(* Logix 5000 project; controller DispersionPlc vendor 1 type 14 code 108 rev 34.11; software revision 34.01; part 18 of 22 *)
(* tags used below, declared in another part *)
   _JISdebug : DINT;
   constant : REAL;
   Estop_Disp : ALIAS FOR Local:3:I.Data.1;
   FilterChangePB : BOOL;
   FIT_4302_1 : AStd_AnalogInput;
   FQIC_4302_11_CurrentTrasferredLb : DINT;
   FQIC_4302_11_Reset : BOOL;
   FQIC_4302_11_TransferSetpoint : DINT;
   FQIC_4302_11_TransferStopValueLb : DINT;
   GenPurp : AStd_GeneralPurp;
   LAH_4302_11 : BOOL;   // Truck Loading Level Alarm High Probe
   LAH_S4352_1 : ALIAS FOR Local:1:I.Data[27].13;
   resetTimer : BOOL;
   ROC_SP : REAL;
   ROC_SP_10min : REAL;
   S4352_Phase_Circulation : AStd_PLI;
   S4352_Phase_Packaging_Transfer : AStd_PLI;
   S4352_Phase_TT_Transfer : AStd_PLI;
   S52TransferCompletePB : BOOL;
   SP : REAL;
   SV_4302_1 : AStd_VlvOC;
   SV_S52_2 : AStd_VlvOC;
   T4302_Phase_S52_Transfer : AStd_PLI;
   T4302_Phase_S52_Transfer_AOI : AStd_PLI_AOI;
   T4302_Phase_TT_Transfer : AStd_PLI;
   T4302_Phase_TT_Transfer_AOI : AStd_PLI_AOI;
   T4302_PhaseAgitation : AStd_PLI;
   T4302_PhaseAgitation_AOI : AStd_PLI_AOI;
   T4302_PhaseTempControl : AStd_PLI;
   T4302_PhaseTempControl_AOI : AStd_PLI_AOI;
   T4302_RampControl : BOOL;
   T4302_RampControl_ONS : BOOL;
   T4302_RampControl_ONS_2 : BOOL;
   T4302_RampControlTOn : TIMER;
   T4302TruckTransferCompletePB : BOOL;
   TCV_4302_1 : AStd_VlvModulating;
   TCV_4302_2 : AStd_VlvModulating;
   TCV_4302_2_Mode : SINT;
   TE_4302A : ALIAS FOR Local:8:I.Ch5Data;
   TempChange : REAL;
   TIC_4302_1 : AStd_PIDInterface;
   TIC_4302_1_AOI : AStd_PIDInterface_AOI;
   TIC_4302_1_PID : PID_ENHANCED;
   TIC_4302_4C : AStd_PIDInterface;
   TIC_4302_4C_AOI : AStd_PIDInterface_AOI;
   TIC_4302_4C_PID : PID_ENHANCED;
   TIC_4302_4H : AStd_PIDInterface;
   TIC_4302_4H_AOI : AStd_PIDInterface_AOI;
   TIC_4302_4H_PID : PID_ENHANCED;
   TIT_4302_1 : AStd_AnalogInput;
   TIT_4302_4 : AStd_AnalogInput;
   VFD_4302_1 : AStd_VFD;
   VFD_P_4302_2 : AStd_VFD;
   WIT_4302_1 : AStd_AnalogInput;
   XV_4302_12 : AStd_VlvOC;
   XV_4302_13 : AStd_VlvOC;
   XV_4302_5 : AStd_VlvOC;
   XV_4302_6 : AStd_VlvOC;
   XV_S52_1 : AStd_VlvOC;
   XV_S52_2 : AStd_VlvOC;
(* Unit_T4302, continued *)

ROUTINE Phase_Agitation   (* ladder *)
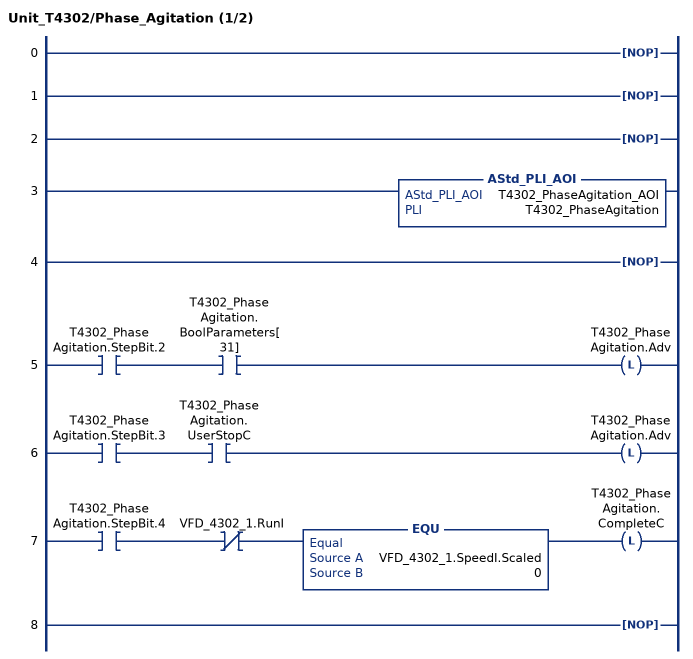
   0: NOP();
   1: NOP();
   2: NOP();
   3: AStd_PLI_AOI(T4302_PhaseAgitation_AOI,T4302_PhaseAgitation);
   4: NOP();
   5: XIC(T4302_PhaseAgitation.StepBit.2)XIC(T4302_PhaseAgitation.BoolParameters[31])OTL(T4302_PhaseAgitation.Adv);
   6: XIC(T4302_PhaseAgitation.StepBit.3)XIC(T4302_PhaseAgitation.UserStopC)OTL(T4302_PhaseAgitation.Adv);
   7: XIC(T4302_PhaseAgitation.StepBit.4)XIO(VFD_4302_1.RunI)EQU(VFD_4302_1.SpeedI.Scaled,0)OTL(T4302_PhaseAgitation.CompleteC);
   8: NOP();
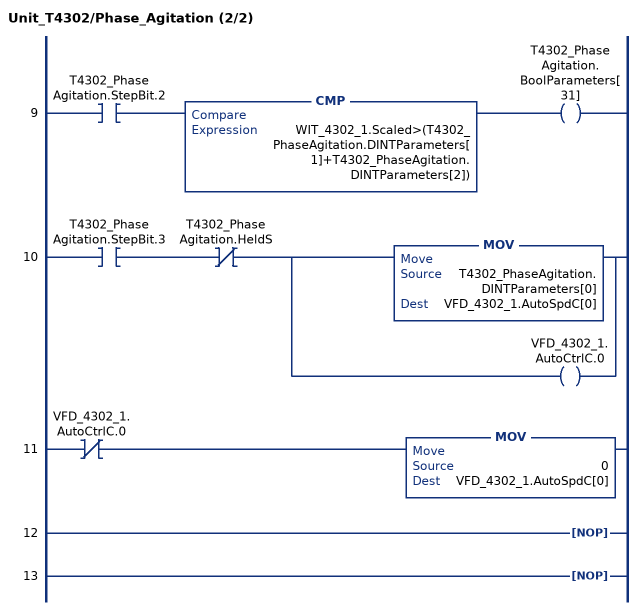
   9: XIC(T4302_PhaseAgitation.StepBit.2)CMP(WIT_4302_1.Scaled>(T4302_PhaseAgitation.DINTParameters[1]+T4302_PhaseAgitation.DINTParameters[2]))OTE(T4302_PhaseAgitation.BoolParameters[31]);
   10: XIC(T4302_PhaseAgitation.StepBit.3)XIO(T4302_PhaseAgitation.HeldS)[MOV(T4302_PhaseAgitation.DINTParameters[0],VFD_4302_1.AutoSpdC[0]) ,OTE(VFD_4302_1.AutoCtrlC.0) ];
   11: XIO(VFD_4302_1.AutoCtrlC.0)MOV(0,VFD_4302_1.AutoSpdC[0]);
   12: NOP();
   13: NOP();
END_ROUTINE

ROUTINE Phase_S52_Transfer   (* ladder *)
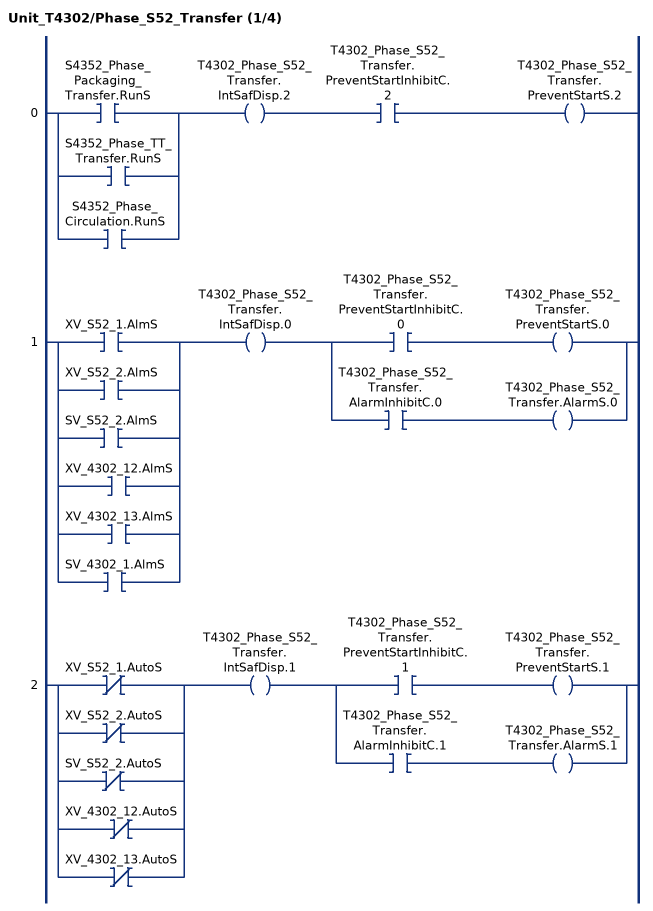
   0: [XIC(S4352_Phase_Packaging_Transfer.RunS) ,XIC(S4352_Phase_TT_Transfer.RunS) ,XIC(S4352_Phase_Circulation.RunS) ]OTE(T4302_Phase_S52_Transfer.IntSafDisp.2)XIC(T4302_Phase_S52_Transfer.PreventStartInhibitC.2)OTE(T4302_Phase_S52_Transfer.PreventStartS.2);
   1: [XIC(XV_S52_1.AlmS) ,XIC(XV_S52_2.AlmS) ,XIC(SV_S52_2.AlmS) ,XIC(XV_4302_12.AlmS) ,XIC(XV_4302_13.AlmS) ,XIC(SV_4302_1.AlmS) ]OTE(T4302_Phase_S52_Transfer.IntSafDisp.0)[XIC(T4302_Phase_S52_Transfer.PreventStartInhibitC.0) OTE(T4302_Phase_S52_Transfer.PreventStartS.0) ,XIC(T4302_Phase_S52_Transfer.AlarmInhibitC.0) OTE(T4302_Phase_S52_Transfer.AlarmS.0) ];
   2: [XIO(XV_S52_1.AutoS) ,XIO(XV_S52_2.AutoS) ,XIO(SV_S52_2.AutoS) ,XIO(XV_4302_12.AutoS) ,XIO(XV_4302_13.AutoS) ]OTE(T4302_Phase_S52_Transfer.IntSafDisp.1)[XIC(T4302_Phase_S52_Transfer.PreventStartInhibitC.1) OTE(T4302_Phase_S52_Transfer.PreventStartS.1) ,XIC(T4302_Phase_S52_Transfer.AlarmInhibitC.1) OTE(T4302_Phase_S52_Transfer.AlarmS.1) ];
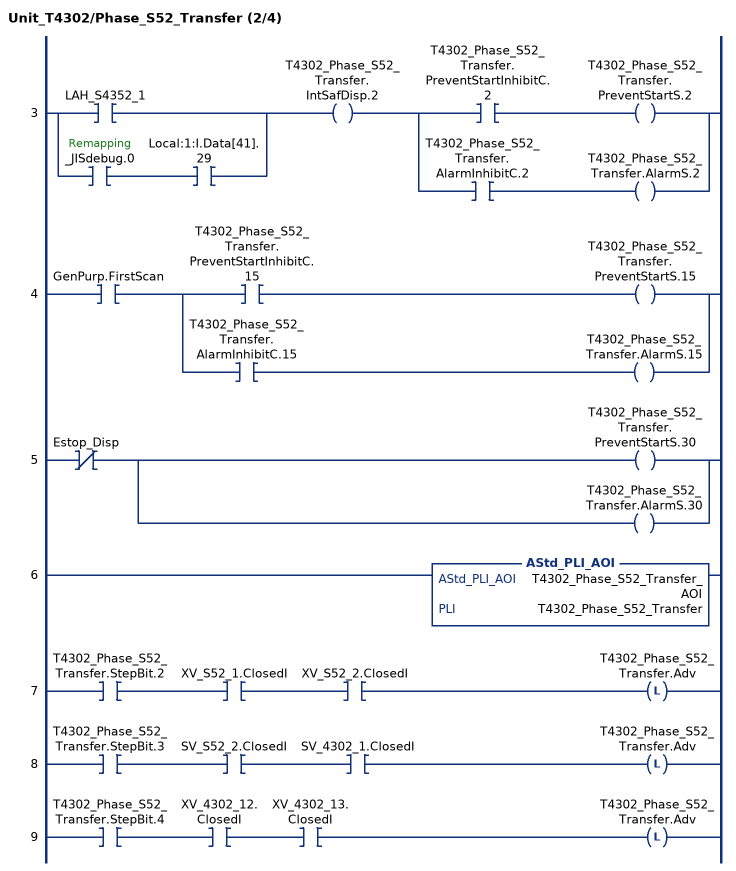
   3: [XIC(LAH_S4352_1) ,XIC(_JISdebug.0) XIC(Local:1:I.Data[41].29) ]OTE(T4302_Phase_S52_Transfer.IntSafDisp.2)[XIC(T4302_Phase_S52_Transfer.PreventStartInhibitC.2) OTE(T4302_Phase_S52_Transfer.PreventStartS.2) ,XIC(T4302_Phase_S52_Transfer.AlarmInhibitC.2) OTE(T4302_Phase_S52_Transfer.AlarmS.2) ];
   4: XIC(GenPurp.FirstScan)[XIC(T4302_Phase_S52_Transfer.PreventStartInhibitC.15) OTE(T4302_Phase_S52_Transfer.PreventStartS.15) ,XIC(T4302_Phase_S52_Transfer.AlarmInhibitC.15) OTE(T4302_Phase_S52_Transfer.AlarmS.15) ];
   5: XIO(Estop_Disp)[OTE(T4302_Phase_S52_Transfer.PreventStartS.30) ,OTE(T4302_Phase_S52_Transfer.AlarmS.30) ];
   6: AStd_PLI_AOI(T4302_Phase_S52_Transfer_AOI,T4302_Phase_S52_Transfer);
   7: XIC(T4302_Phase_S52_Transfer.StepBit.2)XIC(XV_S52_1.ClosedI)XIC(XV_S52_2.ClosedI)OTL(T4302_Phase_S52_Transfer.Adv);
   8: XIC(T4302_Phase_S52_Transfer.StepBit.3)XIC(SV_S52_2.ClosedI)XIC(SV_4302_1.ClosedI)OTL(T4302_Phase_S52_Transfer.Adv);
   9: XIC(T4302_Phase_S52_Transfer.StepBit.4)XIC(XV_4302_12.ClosedI)XIC(XV_4302_13.ClosedI)OTL(T4302_Phase_S52_Transfer.Adv);
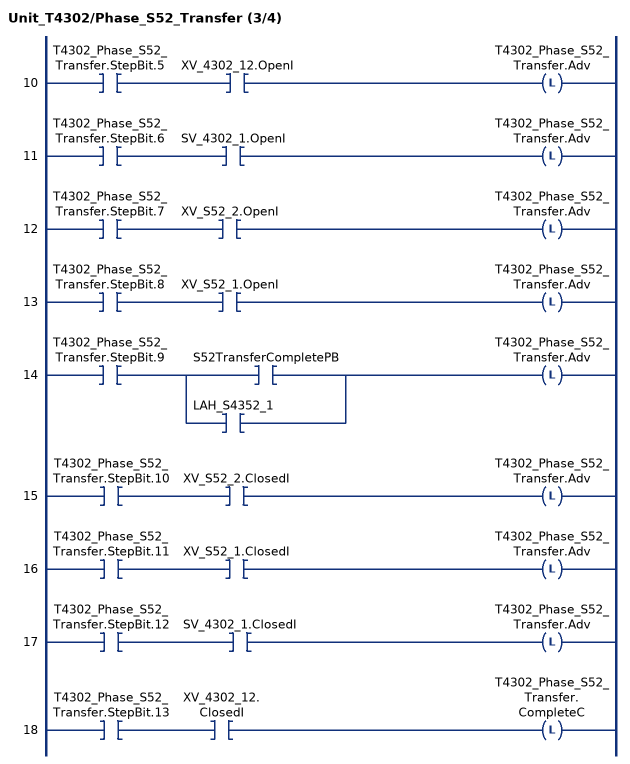
   10: XIC(T4302_Phase_S52_Transfer.StepBit.5)XIC(XV_4302_12.OpenI)OTL(T4302_Phase_S52_Transfer.Adv);
   11: XIC(T4302_Phase_S52_Transfer.StepBit.6)XIC(SV_4302_1.OpenI)OTL(T4302_Phase_S52_Transfer.Adv);
   12: XIC(T4302_Phase_S52_Transfer.StepBit.7)XIC(XV_S52_2.OpenI)OTL(T4302_Phase_S52_Transfer.Adv);
   13: XIC(T4302_Phase_S52_Transfer.StepBit.8)XIC(XV_S52_1.OpenI)OTL(T4302_Phase_S52_Transfer.Adv);
   14: XIC(T4302_Phase_S52_Transfer.StepBit.9)[XIC(S52TransferCompletePB) ,XIC(LAH_S4352_1) ]OTL(T4302_Phase_S52_Transfer.Adv);
   15: XIC(T4302_Phase_S52_Transfer.StepBit.10)XIC(XV_S52_2.ClosedI)OTL(T4302_Phase_S52_Transfer.Adv);
   16: XIC(T4302_Phase_S52_Transfer.StepBit.11)XIC(XV_S52_1.ClosedI)OTL(T4302_Phase_S52_Transfer.Adv);
   17: XIC(T4302_Phase_S52_Transfer.StepBit.12)XIC(SV_4302_1.ClosedI)OTL(T4302_Phase_S52_Transfer.Adv);
   18: XIC(T4302_Phase_S52_Transfer.StepBit.13)XIC(XV_4302_12.ClosedI)OTL(T4302_Phase_S52_Transfer.CompleteC);
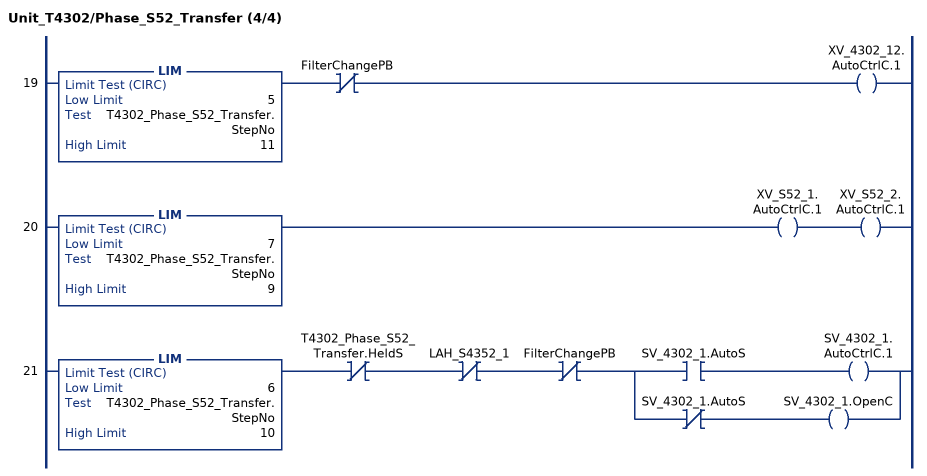
   19: LIM(5,T4302_Phase_S52_Transfer.StepNo,11)XIO(FilterChangePB)OTE(XV_4302_12.AutoCtrlC.1);
   20: LIM(7,T4302_Phase_S52_Transfer.StepNo,9)OTE(XV_S52_1.AutoCtrlC.1)OTE(XV_S52_2.AutoCtrlC.1);
   21: LIM(6,T4302_Phase_S52_Transfer.StepNo,10)XIO(T4302_Phase_S52_Transfer.HeldS)XIO(LAH_S4352_1)XIO(FilterChangePB)[XIC(SV_4302_1.AutoS) OTE(SV_4302_1.AutoCtrlC.1) ,XIO(SV_4302_1.AutoS) OTE(SV_4302_1.OpenC) ];
END_ROUTINE

ROUTINE Phase_TempControl   (* ladder *)
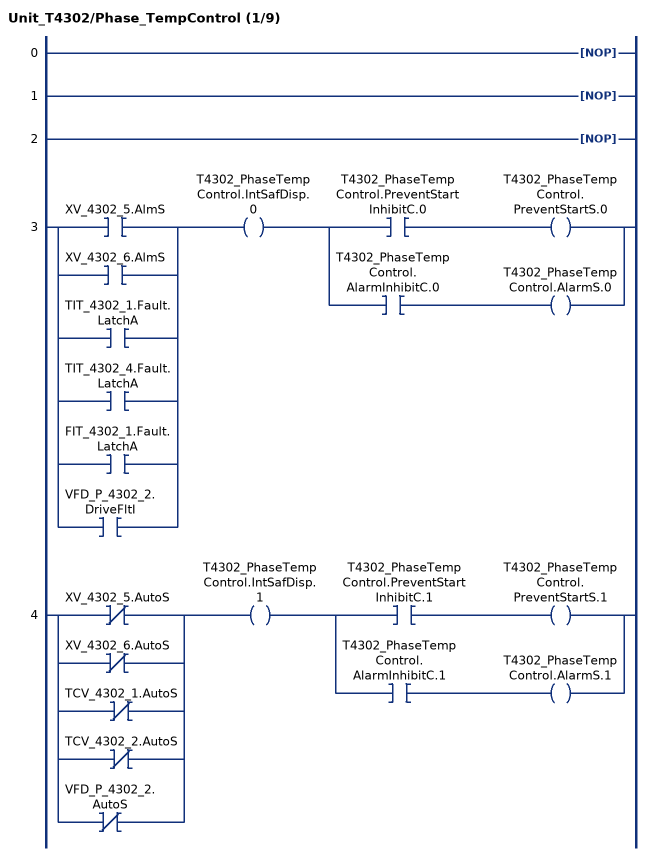
   0: NOP();
   1: NOP();
   2: NOP();
   3: [XIC(XV_4302_5.AlmS) ,XIC(XV_4302_6.AlmS) ,XIC(TIT_4302_1.Fault.LatchA) ,XIC(TIT_4302_4.Fault.LatchA) ,XIC(FIT_4302_1.Fault.LatchA) ,XIC(VFD_P_4302_2.DriveFltI) ]OTE(T4302_PhaseTempControl.IntSafDisp.0)[XIC(T4302_PhaseTempControl.PreventStartInhibitC.0) OTE(T4302_PhaseTempControl.PreventStartS.0) ,XIC(T4302_PhaseTempControl.AlarmInhibitC.0) OTE(T4302_PhaseTempControl.AlarmS.0) ];
   4: [XIO(XV_4302_5.AutoS) ,XIO(XV_4302_6.AutoS) ,XIO(TCV_4302_1.AutoS) ,XIO(TCV_4302_2.AutoS) ,XIO(VFD_P_4302_2.AutoS) ]OTE(T4302_PhaseTempControl.IntSafDisp.1)[XIC(T4302_PhaseTempControl.PreventStartInhibitC.1) OTE(T4302_PhaseTempControl.PreventStartS.1) ,XIC(T4302_PhaseTempControl.AlarmInhibitC.1) OTE(T4302_PhaseTempControl.AlarmS.1) ];
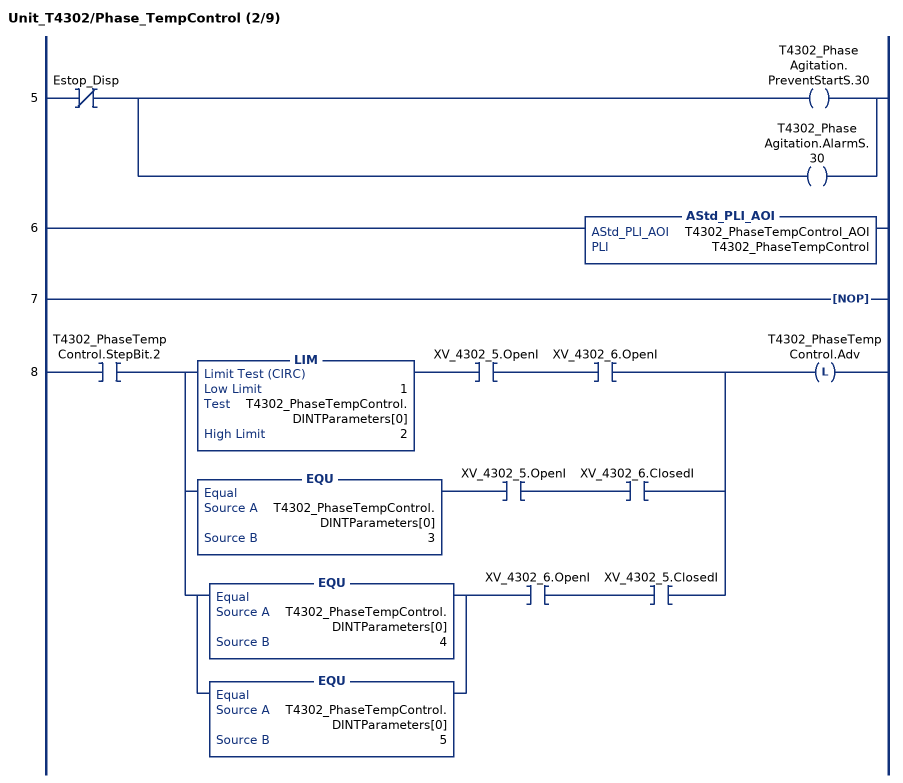
   5: XIO(Estop_Disp)[OTE(T4302_PhaseAgitation.PreventStartS.30) ,OTE(T4302_PhaseAgitation.AlarmS.30) ];
   6: AStd_PLI_AOI(T4302_PhaseTempControl_AOI,T4302_PhaseTempControl);
   7: NOP();
   8: XIC(T4302_PhaseTempControl.StepBit.2)[LIM(1,T4302_PhaseTempControl.DINTParameters[0],2) XIC(XV_4302_5.OpenI) XIC(XV_4302_6.OpenI) ,EQU(T4302_PhaseTempControl.DINTParameters[0],3) XIC(XV_4302_5.OpenI) XIC(XV_4302_6.ClosedI) ,[EQU(T4302_PhaseTempControl.DINTParameters[0],4) ,EQU(T4302_PhaseTempControl.DINTParameters[0],5) ] XIC(XV_4302_6.OpenI) XIC(XV_4302_5.ClosedI) ]OTL(T4302_PhaseTempControl.Adv);
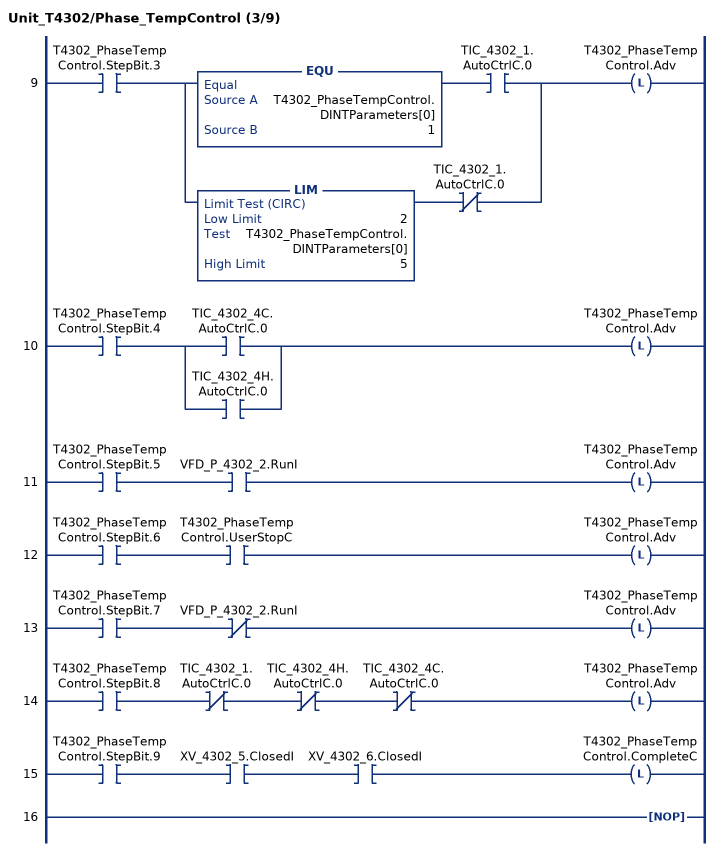
   9: XIC(T4302_PhaseTempControl.StepBit.3)[EQU(T4302_PhaseTempControl.DINTParameters[0],1) XIC(TIC_4302_1.AutoCtrlC.0) ,LIM(2,T4302_PhaseTempControl.DINTParameters[0],5) XIO(TIC_4302_1.AutoCtrlC.0) ]OTL(T4302_PhaseTempControl.Adv);
   10: XIC(T4302_PhaseTempControl.StepBit.4)[XIC(TIC_4302_4C.AutoCtrlC.0) ,XIC(TIC_4302_4H.AutoCtrlC.0) ]OTL(T4302_PhaseTempControl.Adv);
   11: XIC(T4302_PhaseTempControl.StepBit.5)XIC(VFD_P_4302_2.RunI)OTL(T4302_PhaseTempControl.Adv);
   12: XIC(T4302_PhaseTempControl.StepBit.6)XIC(T4302_PhaseTempControl.UserStopC)OTL(T4302_PhaseTempControl.Adv);
   13: XIC(T4302_PhaseTempControl.StepBit.7)XIO(VFD_P_4302_2.RunI)OTL(T4302_PhaseTempControl.Adv);
   14: XIC(T4302_PhaseTempControl.StepBit.8)XIO(TIC_4302_1.AutoCtrlC.0)XIO(TIC_4302_4H.AutoCtrlC.0)XIO(TIC_4302_4C.AutoCtrlC.0)OTL(T4302_PhaseTempControl.Adv);
   15: XIC(T4302_PhaseTempControl.StepBit.9)XIC(XV_4302_5.ClosedI)XIC(XV_4302_6.ClosedI)OTL(T4302_PhaseTempControl.CompleteC);
   16: NOP();
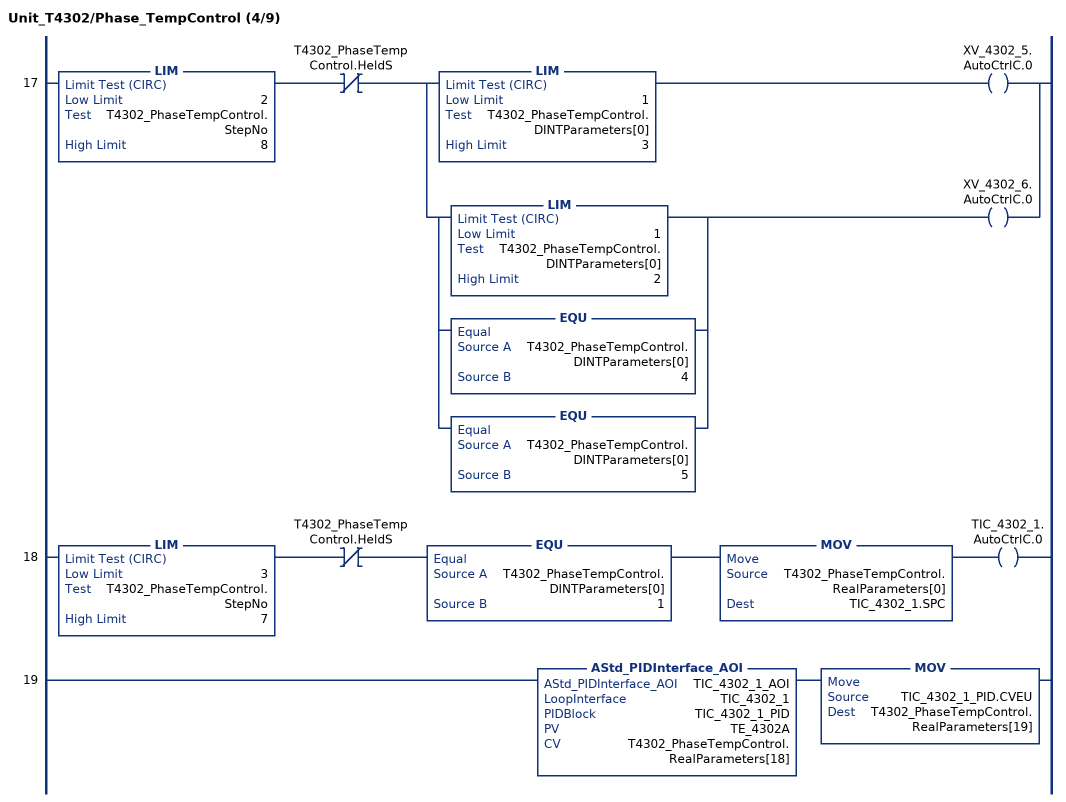
   17: LIM(2,T4302_PhaseTempControl.StepNo,8)XIO(T4302_PhaseTempControl.HeldS)[LIM(1,T4302_PhaseTempControl.DINTParameters[0],3) OTE(XV_4302_5.AutoCtrlC.0) ,[LIM(1,T4302_PhaseTempControl.DINTParameters[0],2) ,[EQU(T4302_PhaseTempControl.DINTParameters[0],4) ,EQU(T4302_PhaseTempControl.DINTParameters[0],5) ] ] OTE(XV_4302_6.AutoCtrlC.0) ];
   18: LIM(3,T4302_PhaseTempControl.StepNo,7)XIO(T4302_PhaseTempControl.HeldS)EQU(T4302_PhaseTempControl.DINTParameters[0],1)MOV(T4302_PhaseTempControl.RealParameters[0],TIC_4302_1.SPC)OTE(TIC_4302_1.AutoCtrlC.0);
   19: AStd_PIDInterface_AOI(TIC_4302_1_AOI,TIC_4302_1,TIC_4302_1_PID,TE_4302A,T4302_PhaseTempControl.RealParameters[18])MOV(TIC_4302_1_PID.CVEU,T4302_PhaseTempControl.RealParameters[19]);
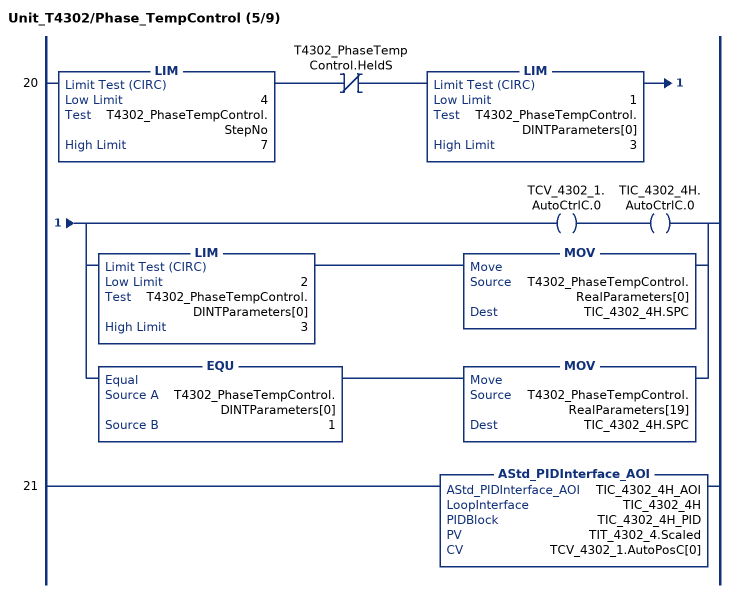
   20: LIM(4,T4302_PhaseTempControl.StepNo,7)XIO(T4302_PhaseTempControl.HeldS)LIM(1,T4302_PhaseTempControl.DINTParameters[0],3)[OTE(TCV_4302_1.AutoCtrlC.0) OTE(TIC_4302_4H.AutoCtrlC.0) ,LIM(2,T4302_PhaseTempControl.DINTParameters[0],3) MOV(T4302_PhaseTempControl.RealParameters[0],TIC_4302_4H.SPC) ,EQU(T4302_PhaseTempControl.DINTParameters[0],1) MOV(T4302_PhaseTempControl.RealParameters[19],TIC_4302_4H.SPC) ];
   21: AStd_PIDInterface_AOI(TIC_4302_4H_AOI,TIC_4302_4H,TIC_4302_4H_PID,TIT_4302_4.Scaled,TCV_4302_1.AutoPosC[0]);
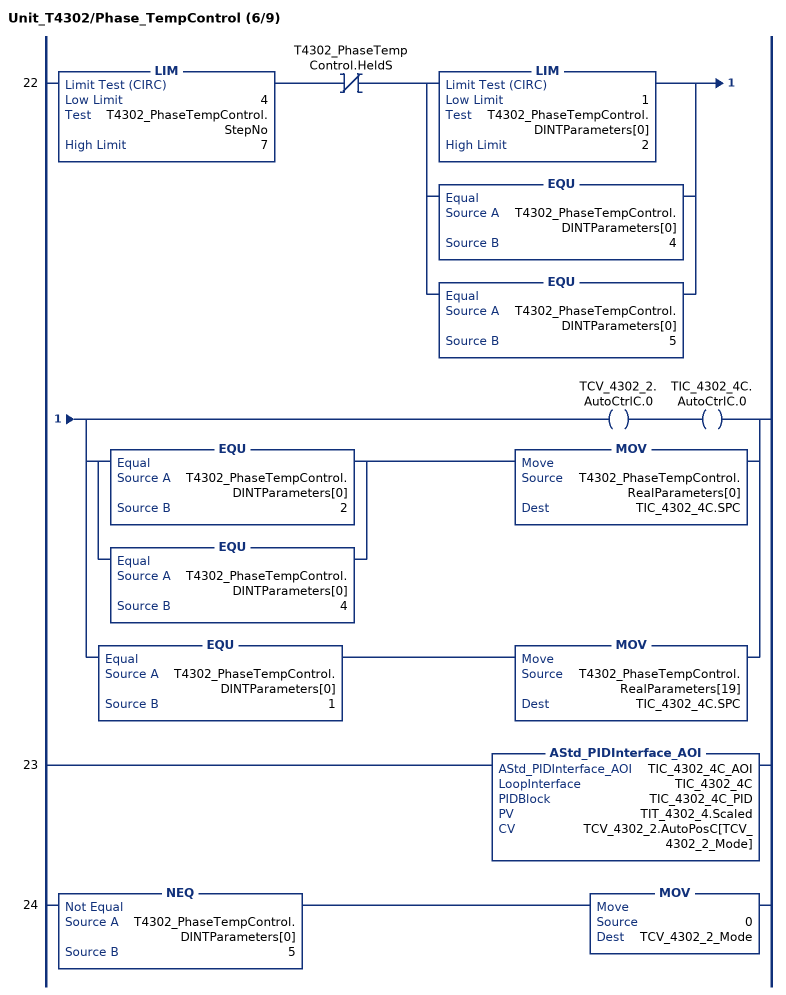
   22: LIM(4,T4302_PhaseTempControl.StepNo,7)XIO(T4302_PhaseTempControl.HeldS)[LIM(1,T4302_PhaseTempControl.DINTParameters[0],2) ,[EQU(T4302_PhaseTempControl.DINTParameters[0],4) ,EQU(T4302_PhaseTempControl.DINTParameters[0],5) ] ][OTE(TCV_4302_2.AutoCtrlC.0) OTE(TIC_4302_4C.AutoCtrlC.0) ,[EQU(T4302_PhaseTempControl.DINTParameters[0],2) ,EQU(T4302_PhaseTempControl.DINTParameters[0],4) ] MOV(T4302_PhaseTempControl.RealParameters[0],TIC_4302_4C.SPC) ,EQU(T4302_PhaseTempControl.DINTParameters[0],1) MOV(T4302_PhaseTempControl.RealParameters[19],TIC_4302_4C.SPC) ];
   23: AStd_PIDInterface_AOI(TIC_4302_4C_AOI,TIC_4302_4C,TIC_4302_4C_PID,TIT_4302_4.Scaled,TCV_4302_2.AutoPosC[TCV_4302_2_Mode]);
   24: NEQ(T4302_PhaseTempControl.DINTParameters[0],5)MOV(0,TCV_4302_2_Mode);
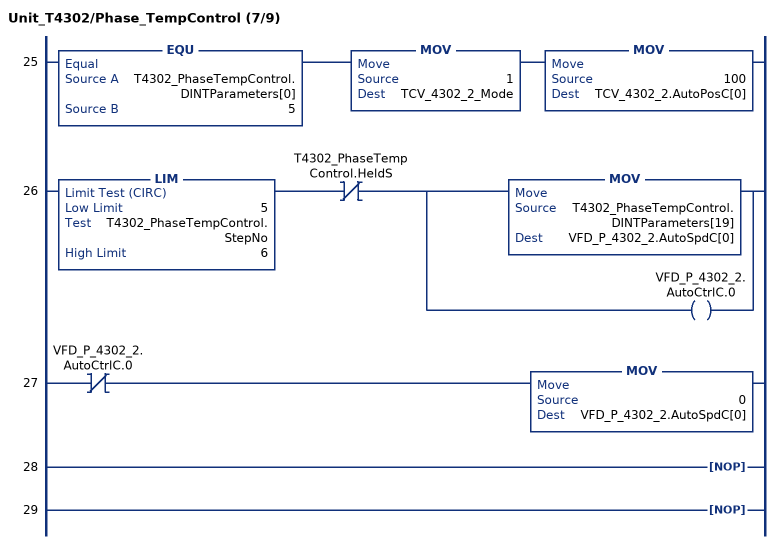
   25: EQU(T4302_PhaseTempControl.DINTParameters[0],5)MOV(1,TCV_4302_2_Mode)MOV(100,TCV_4302_2.AutoPosC[0]);
   26: LIM(5,T4302_PhaseTempControl.StepNo,6)XIO(T4302_PhaseTempControl.HeldS)[MOV(T4302_PhaseTempControl.DINTParameters[19],VFD_P_4302_2.AutoSpdC[0]) ,OTE(VFD_P_4302_2.AutoCtrlC.0) ];
   27: XIO(VFD_P_4302_2.AutoCtrlC.0)MOV(0,VFD_P_4302_2.AutoSpdC[0]);
   28: NOP();
   29: NOP();
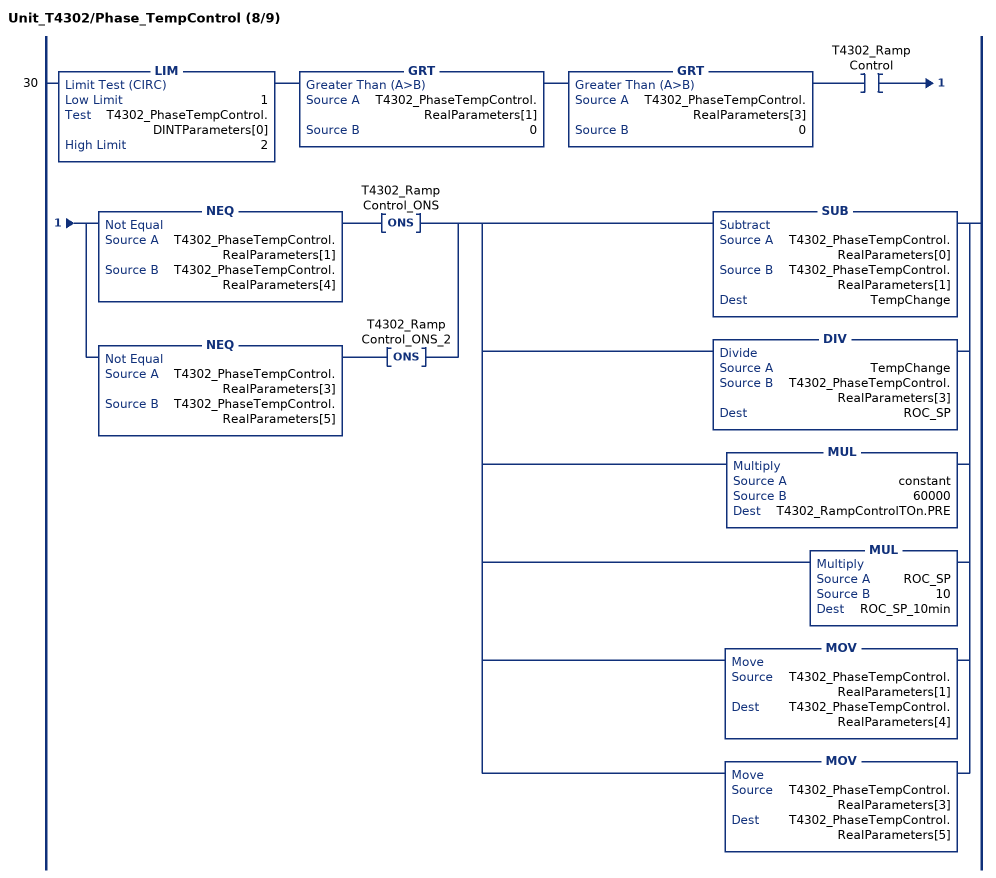
   30: LIM(1,T4302_PhaseTempControl.DINTParameters[0],2)GRT(T4302_PhaseTempControl.RealParameters[1],0)GRT(T4302_PhaseTempControl.RealParameters[3],0)XIC(T4302_RampControl)[NEQ(T4302_PhaseTempControl.RealParameters[1],T4302_PhaseTempControl.RealParameters[4]) ONS(T4302_RampControl_ONS) ,NEQ(T4302_PhaseTempControl.RealParameters[3],T4302_PhaseTempControl.RealParameters[5]) ONS(T4302_RampControl_ONS_2) ][SUB(T4302_PhaseTempControl.RealParameters[0],T4302_PhaseTempControl.RealParameters[1],TempChange) ,DIV(TempChange,T4302_PhaseTempControl.RealParameters[3],ROC_SP) ,MUL(constant,60000,T4302_RampControlTOn.PRE) ,MUL(ROC_SP,10,ROC_SP_10min) ,MOV(T4302_PhaseTempControl.RealParameters[1],T4302_PhaseTempControl.RealParameters[4]) ,MOV(T4302_PhaseTempControl.RealParameters[3],T4302_PhaseTempControl.RealParameters[5]) ];
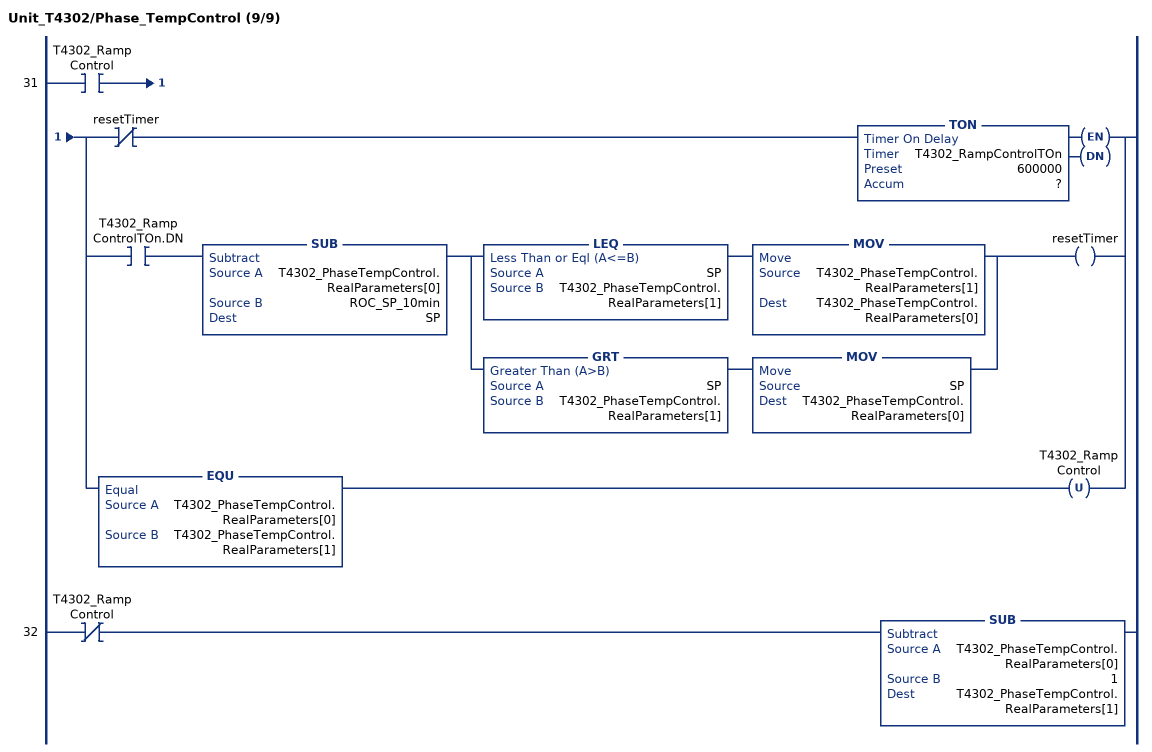
   31: XIC(T4302_RampControl)[XIO(resetTimer) TON(T4302_RampControlTOn,?,?) ,[XIC(T4302_RampControlTOn.DN) SUB(T4302_PhaseTempControl.RealParameters[0],ROC_SP_10min,SP) [LEQ(SP,T4302_PhaseTempControl.RealParameters[1]) MOV(T4302_PhaseTempControl.RealParameters[1],T4302_PhaseTempControl.RealParameters[0]) ,GRT(SP,T4302_PhaseTempControl.RealParameters[1]) MOV(SP,T4302_PhaseTempControl.RealParameters[0]) ] OTE(resetTimer) ,EQU(T4302_PhaseTempControl.RealParameters[0],T4302_PhaseTempControl.RealParameters[1]) OTU(T4302_RampControl) ] ];
   32: XIO(T4302_RampControl)SUB(T4302_PhaseTempControl.RealParameters[0],1,T4302_PhaseTempControl.RealParameters[1]);
END_ROUTINE

ROUTINE Phase_TT_Transfer   (* ladder *)
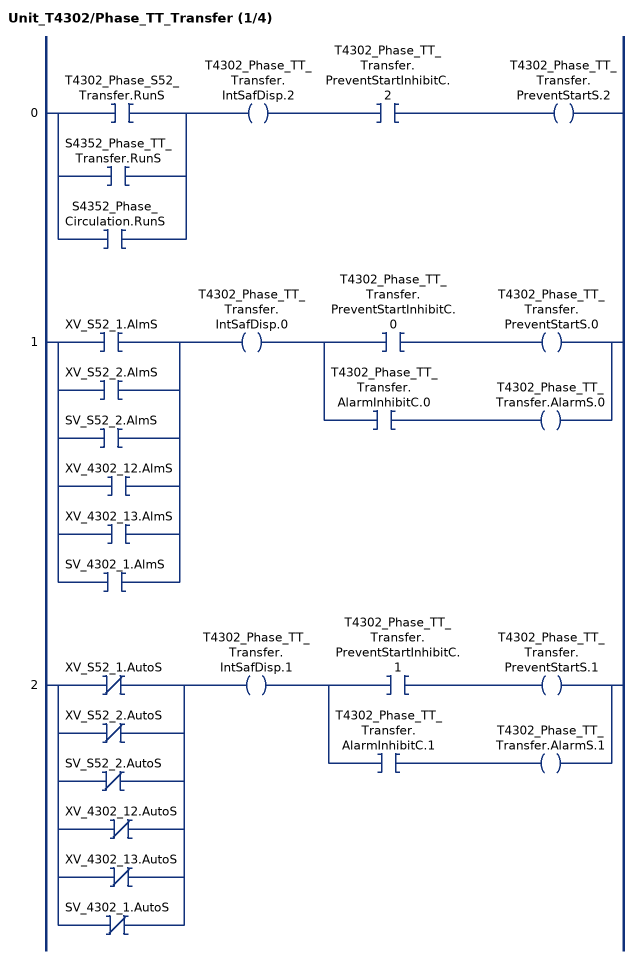
   0: [XIC(T4302_Phase_S52_Transfer.RunS) ,XIC(S4352_Phase_TT_Transfer.RunS) ,XIC(S4352_Phase_Circulation.RunS) ]OTE(T4302_Phase_TT_Transfer.IntSafDisp.2)XIC(T4302_Phase_TT_Transfer.PreventStartInhibitC.2)OTE(T4302_Phase_TT_Transfer.PreventStartS.2);
   1: [XIC(XV_S52_1.AlmS) ,XIC(XV_S52_2.AlmS) ,XIC(SV_S52_2.AlmS) ,XIC(XV_4302_12.AlmS) ,XIC(XV_4302_13.AlmS) ,XIC(SV_4302_1.AlmS) ]OTE(T4302_Phase_TT_Transfer.IntSafDisp.0)[XIC(T4302_Phase_TT_Transfer.PreventStartInhibitC.0) OTE(T4302_Phase_TT_Transfer.PreventStartS.0) ,XIC(T4302_Phase_TT_Transfer.AlarmInhibitC.0) OTE(T4302_Phase_TT_Transfer.AlarmS.0) ];
   2: [XIO(XV_S52_1.AutoS) ,XIO(XV_S52_2.AutoS) ,XIO(SV_S52_2.AutoS) ,XIO(XV_4302_12.AutoS) ,XIO(XV_4302_13.AutoS) ,XIO(SV_4302_1.AutoS) ]OTE(T4302_Phase_TT_Transfer.IntSafDisp.1)[XIC(T4302_Phase_TT_Transfer.PreventStartInhibitC.1) OTE(T4302_Phase_TT_Transfer.PreventStartS.1) ,XIC(T4302_Phase_TT_Transfer.AlarmInhibitC.1) OTE(T4302_Phase_TT_Transfer.AlarmS.1) ];
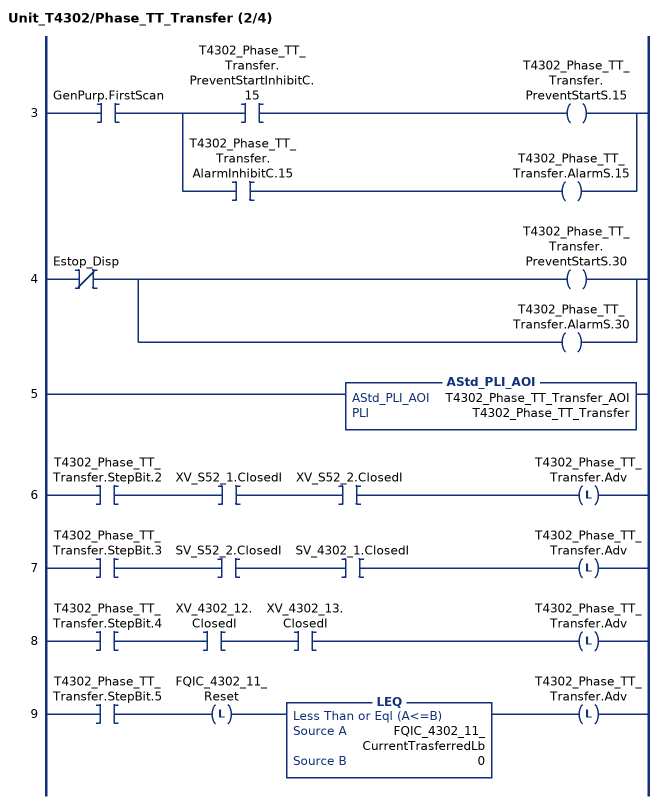
   3: XIC(GenPurp.FirstScan)[XIC(T4302_Phase_TT_Transfer.PreventStartInhibitC.15) OTE(T4302_Phase_TT_Transfer.PreventStartS.15) ,XIC(T4302_Phase_TT_Transfer.AlarmInhibitC.15) OTE(T4302_Phase_TT_Transfer.AlarmS.15) ];
   4: XIO(Estop_Disp)[OTE(T4302_Phase_TT_Transfer.PreventStartS.30) ,OTE(T4302_Phase_TT_Transfer.AlarmS.30) ];
   5: AStd_PLI_AOI(T4302_Phase_TT_Transfer_AOI,T4302_Phase_TT_Transfer);
   6: XIC(T4302_Phase_TT_Transfer.StepBit.2)XIC(XV_S52_1.ClosedI)XIC(XV_S52_2.ClosedI)OTL(T4302_Phase_TT_Transfer.Adv);
   7: XIC(T4302_Phase_TT_Transfer.StepBit.3)XIC(SV_S52_2.ClosedI)XIC(SV_4302_1.ClosedI)OTL(T4302_Phase_TT_Transfer.Adv);
   8: XIC(T4302_Phase_TT_Transfer.StepBit.4)XIC(XV_4302_12.ClosedI)XIC(XV_4302_13.ClosedI)OTL(T4302_Phase_TT_Transfer.Adv);
   9: XIC(T4302_Phase_TT_Transfer.StepBit.5)OTL(FQIC_4302_11_Reset)LEQ(FQIC_4302_11_CurrentTrasferredLb,0)OTL(T4302_Phase_TT_Transfer.Adv);
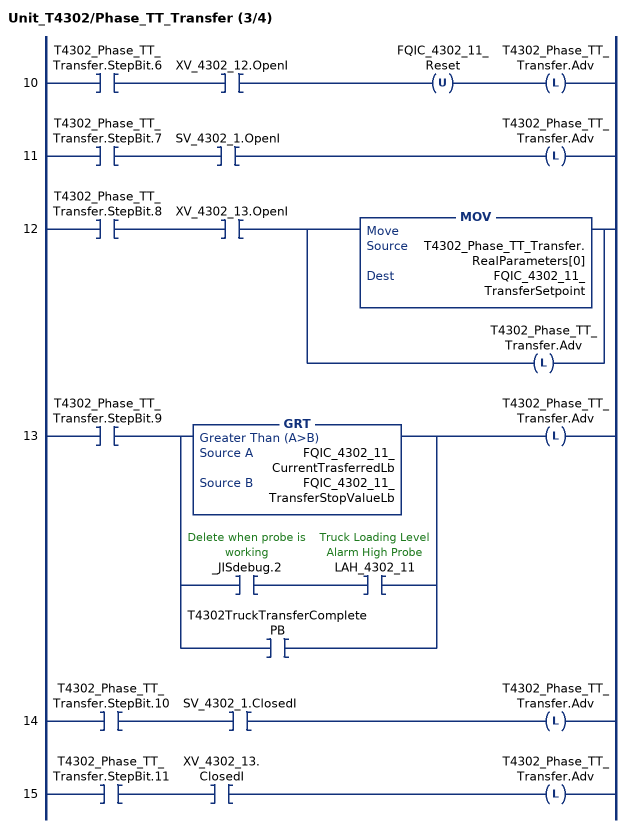
   10: XIC(T4302_Phase_TT_Transfer.StepBit.6)XIC(XV_4302_12.OpenI)OTU(FQIC_4302_11_Reset)OTL(T4302_Phase_TT_Transfer.Adv);
   11: XIC(T4302_Phase_TT_Transfer.StepBit.7)XIC(SV_4302_1.OpenI)OTL(T4302_Phase_TT_Transfer.Adv);
   12: XIC(T4302_Phase_TT_Transfer.StepBit.8)XIC(XV_4302_13.OpenI)[MOV(T4302_Phase_TT_Transfer.RealParameters[0],FQIC_4302_11_TransferSetpoint) ,OTL(T4302_Phase_TT_Transfer.Adv) ];
   13: XIC(T4302_Phase_TT_Transfer.StepBit.9)[GRT(FQIC_4302_11_CurrentTrasferredLb,FQIC_4302_11_TransferStopValueLb) ,XIC(_JISdebug.2) XIC(LAH_4302_11) ,XIC(T4302TruckTransferCompletePB) ]OTL(T4302_Phase_TT_Transfer.Adv);
   14: XIC(T4302_Phase_TT_Transfer.StepBit.10)XIC(SV_4302_1.ClosedI)OTL(T4302_Phase_TT_Transfer.Adv);
   15: XIC(T4302_Phase_TT_Transfer.StepBit.11)XIC(XV_4302_13.ClosedI)OTL(T4302_Phase_TT_Transfer.Adv);
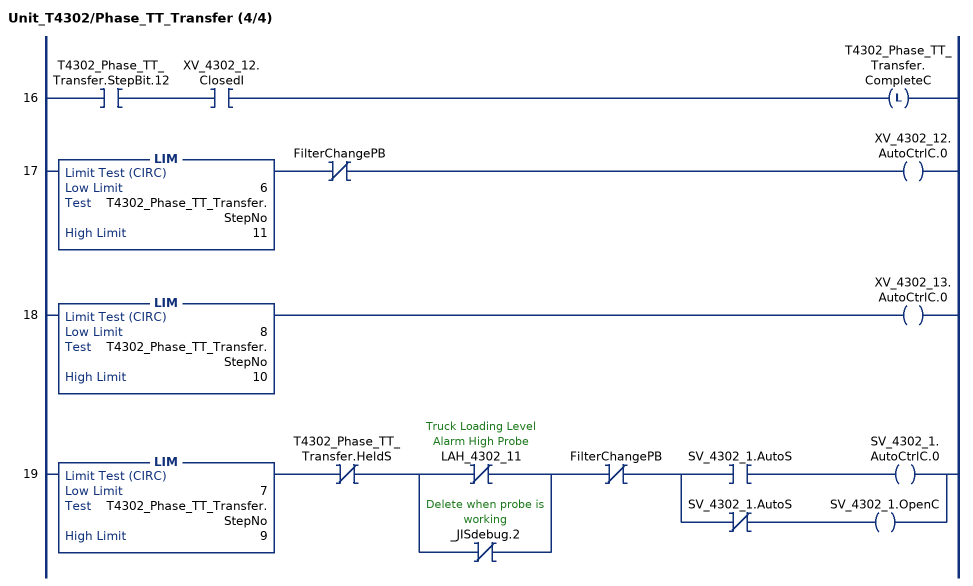
   16: XIC(T4302_Phase_TT_Transfer.StepBit.12)XIC(XV_4302_12.ClosedI)OTL(T4302_Phase_TT_Transfer.CompleteC);
   17: LIM(6,T4302_Phase_TT_Transfer.StepNo,11)XIO(FilterChangePB)OTE(XV_4302_12.AutoCtrlC.0);
   18: LIM(8,T4302_Phase_TT_Transfer.StepNo,10)OTE(XV_4302_13.AutoCtrlC.0);
   19: LIM(7,T4302_Phase_TT_Transfer.StepNo,9)XIO(T4302_Phase_TT_Transfer.HeldS)[XIO(LAH_4302_11) ,XIO(_JISdebug.2) ]XIO(FilterChangePB)[XIC(SV_4302_1.AutoS) OTE(SV_4302_1.AutoCtrlC.0) ,XIO(SV_4302_1.AutoS) OTE(SV_4302_1.OpenC) ];
END_ROUTINE
